		MoveL Blend_7396, v5, z10, pHeader\WObj:=wobj0;
		MoveL Blend_7397, v10, z10, pHeader\WObj:=wobj0;
		MoveL Blend_7398, v20, z10, pHeader\WObj:=wobj0;
		MoveL Blend_7399, v10, z10, pHeader\WObj:=wobj0;
	ENDPROC

ENDMODULE
